TYPE
    Data :
    STRUCT
        IncrementDouble : REAL;
		IncrementInt : INT;
		
		DoubleValue:REAL;
		IntValue : INT;
		Recipe : STRING;
    END_STRUCT
END_TYPE

(* stored: Version 1.1.0.1, ProductVersion 3.1.4024.9
   DUT Data: Id {7181b1b0-2451-4466-9693-7d343269a9e0} *)
